// TIA Portal V21 export
FUNCTION "Loadcell_Profinet" : Void   // FC37, LAD
{ S7_Optimized_Access := 'TRUE' }
// stored: SetENOAutomatically false
BEGIN

REGION Network 1: LoadcellCV15
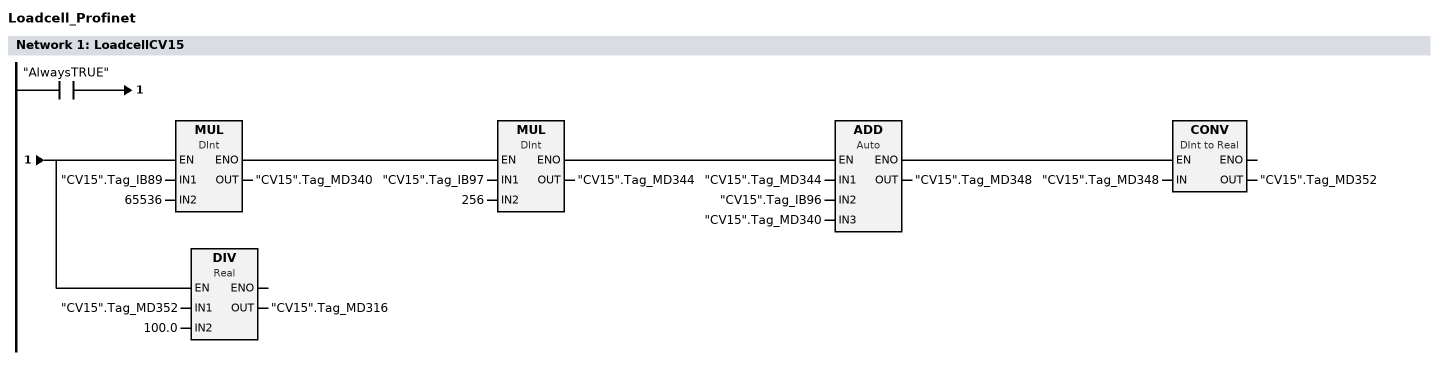
   RUNG wire#powerrail
      Contact( "AlwaysTRUE" )
      wire#w1
      { S7_Templates := "SrcType := DInt" } Mul(in1 := "CV15".Tag_IB89, in2 := 65536, out => "CV15".Tag_MD340)
      { S7_Templates := "SrcType := DInt" } Mul(in1 := "CV15".Tag_IB97, in2 := 256, out => "CV15".Tag_MD344)
      Add(in1 := "CV15".Tag_MD344, in2 := "CV15".Tag_IB96, in3 := "CV15".Tag_MD340, out => "CV15".Tag_MD348)
      { S7_Templates := "[SrcType := DInt, DestType := Real]" } Convert(in := "CV15".Tag_MD348, out => "CV15".Tag_MD352)
   END_RUNG
   RUNG wire#w1
      { S7_Templates := "SrcType := Real" } Div(in1 := "CV15".Tag_MD352, in2 := 100.0, out => "CV15".Tag_MD316)
   END_RUNG
   // the same network as SCL:
   IF "AlwaysTRUE" THEN
       "CV15".Tag_MD340 := "CV15".Tag_IB89 * 65536;
       "CV15".Tag_MD344 := "CV15".Tag_IB97 * 256;
       "CV15".Tag_MD348 := "CV15".Tag_MD344 + "CV15".Tag_IB96 + "CV15".Tag_MD340;
       "CV15".Tag_MD352 := DINT_TO_REAL("CV15".Tag_MD348);
       "CV15".Tag_MD316 := "CV15".Tag_MD352 / 100.0;
   END_IF;
END_REGION
END_FUNCTION
